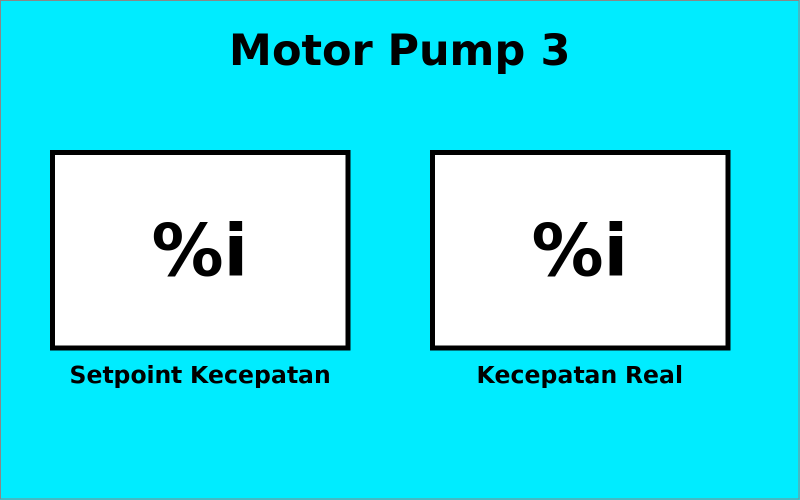
VISUALIZATION Screen_2_Sub_7  // 800x500
    Rectangle (0,0 800x500)
    Label (0,0 800x100), "Motor Pump 3"
    Rectangle (50,150 300x200), "%i", text variable: GVL.HMI_Motor_Pump_3_Input
        OnMouseClick: write GVL.HMI_Motor_Pump_3_Input via VisuDialogs.Numpad
    Label (50,350 300x50), "Setpoint Kecepatan"
    Label (430,350 300x50), "Kecepatan Real"
    Rectangle (430,150 300x200), "%i", text variable: GVL.HMI_Motor_Pump_3_Real
END_VISUALIZATION

(* stored: Version 1.1.0.1, ProductVersion 3.1.4024.12
   Visu Screen_2_Sub_7: Id {7f3f57be-7f10-4ad4-9ca6-d3f316e6eaf0} *)
